{attribute 'GeneratedUsingTerminal: EK1122-0000-0018'}
{attribute addProperty BoxType "EK1122-0000-0018"}
{attribute addProperty Id "A_0060_AT2020_0250_0019_AT2020_0250A_0060_AT2020_0250_0019_AT2020_0250_BB71669A80Beckhoff_AT2xxxsub_EK1100EK1100_AB5A94672A_0001_AT2000_0233_0022AT2000_0D5D20CF80A_0002_AT2000_0233_0023AT2000_0D5D20CF80A_0003_AT2000_0233_0024AT2000_0D5D20CF80A_0004_AT2000_0250_0016AT2000_86175B4184A_0005_AT2000_0250_0017AT2000_86175B4184A_0006_AT2000_0250_0018AT2000_86175B4184A_0007_AT2000_0250_0019AT2000_86175B4184A_0008_AT2000_0250_0020AT2000_86175B4184A_0009_AT2000_0250_0021AT2000_86175B4184A_0010_AT2000_0250_0022AT2000_86175B4184A_0011_AT2000_0250_0023AT2000_86175B4184A_0012_AT2001_0250_0016AT2001_86175B4184A_0013_AT2001_0250_0017AT2001_86175B4184A_0014_AT2001_0250_0018AT2001_86175B4184A_0015_AT2001_0250_0019AT2001_86175B4184A_0016_AT2001_0250_0020AT2001_86175B4184A_0017_AT2001_0250_0022AT2001_86175B4184A_0018_AT2001_0250_0023AT2001_86175B4184A_0019_AT2001_0250_0024AT2001_86175B4184A_0020_AT2002_0249_0021AT2002_86175B4184A_0021_AT2002_0249_0022AT2002_86175B4184A_0022_AT2002_0249_0023AT2002_86175B4184A_0023_AT2002_0250_0022AT2002_86175B4184A_0024_AT2002_0250_0023AT2002_86175B4184A_0025_AT2002_0250_0024AT2002_86175B4184A_0026_AT2020_0250_0018AT2020_86175B4184A_0027_AT2020_0250_0021AT2020_86175B4184A_0028_AT2021_0250_0018AT2021_86175B4184A_0029_AT2021_0250_0020AT2021_86175B4184A_0030_AT2025_0250_0018AT2025_86175B4184A_0031_AT2026_0250_0021AT2026_86175B4184A_0032_AT2026_0250_0023AT2026_86175B4184A_0033_AT2040_0250_0018AT2040_86175B4184A_0034_AT2040_0250_0019AT2040_86175B4184A_0035_AT2040_0250_0020AT2040_86175B4184A_0036_AT2040_0250_0021A_0036_AT2040_0250_0021_991DCE0880A_0037_AT2040_0250_0022A_0037_AT2040_0250_0022_91A22A2880A_0038_AT2040_0250_0023A_0038_AT2040_0250_0023_51A62EE080A_0039_AT2040_0250_0024A_0039_AT2040_0250_0024_A5C6BC0680A_0040_AT2041_0250_0018A_0040_AT2041_0250_0018_C1FAE41E80A_0041_AT2041_0250_0019A_0041_AT2041_0250_0019_61D0A4BA80A_0042_AT2041_0250_0020A_0042_AT2041_0250_0020_CCFA41F280A_0043_AT2041_0250_0021A_0043_AT2041_0250_0021_389AD31480A_0044_AT2041_0250_0022A_0044_AT2041_0250_0022_C805DD5680A_0045_AT2041_0250_0023A_0045_AT2041_0250_0023_C359864080A_0046_AT2042_0250_0024A_0046_AT2042_0250_0024_89BF2BDD80A_0047_AT2050_0500_0016A_0047_AT2050_0500_0016_8100CFFD80A_0048_AT2050_0500_0017A_0048_AT2050_0500_0017_AD089BAB80A_0049_AT2050_0500_0018A_0049_AT2050_0500_0018_5979B14480A_0050_AT2050_0500_0019A_0050_AT2050_0500_0019_873C4A8380A_0051_AT2050_0500_0020A_0051_AT2050_0500_0020_09CCFFA280A_0052_AT2050_0500_0021A_0052_AT2050_0500_0021_D789046580A_0053_AT2050_0500_0022A_0053_AT2050_0500_0022_D1A4391280A_0054_AT2050_0500_0023A_0054_AT2050_0500_0023_206D3BB980A_0055_AT2050_0500_0024A_0055_AT2050_0500_0024_1FDD446180A_0056_AT2050_0501_0017A_0056_AT2050_0501_0017_33D5103780A_0057_AT2050_0501_0020A_0057_AT2050_0501_0020_3B6AF41780A_0058_AT2050_0501_0021A_0058_AT2050_0501_0021_4F11F47C80A_0061_AT2020_0250_0023_AT2020_0250A_0061_AT2020_0250_0023_AT2020_0250_BF05573080A_0062_AT2025_0250_0020_AT2025_0250A_0062_AT2025_0250_0020_AT2025_0250_1F2F179480A_0063_AT2025_0250_0022_AT2025_0250A_0063_AT2025_0250_0022_AT2025_0250_7A10824E80A_0064_AT2025_0250_0023_AT2025_0250A_0064_AT2025_0250_0023_AT2025_0250_1BD08B3080A_0065_AT2026_0250_0019_AT2026_0250A_0065_AT2026_0250_0019_AT2026_0250_37D8DF6680A_0066_AT2026_0250_0020_AT2026_0250A_0066_AT2026_0250_0020_AT2026_0250_3F673B4680A_0067_AT2026_0250_0022_AT2026_0250A_0067_AT2026_0250_0022_AT2026_0250_2DED6B0A80A_0068_AT2026_0250_0024_AT2026_0250A_0068_AT2026_0250_0024_AT2026_0250_E35FF58980A_0069_AT2050_0501_0019_AT2050_0501A_0069_AT2050_0501_0019_AT2050_0501_82BABB4A80A_0070_AT2050_0501_0022_AT2050_0501A_0070_AT2050_0501_0022_AT2050_0501_76DA29AC80A_0071_AT2050_0501_0023_AT2050_0501A_0071_AT2050_0501_0023_AT2050_0501_3753726880A_0072_AT2050_0501_0024_AT2050_0501A_0072_AT2050_0501_0024_AT2050_0501_977932CC80"}
{attribute addProperty CRC "2549082078"}
{attribute addProperty Size "5810"}
TYPE Beckhoff_AT2xxxEK1122_97EFE7DE EXTENDS EK1122_AB5A9467 :
STRUCT
	{attribute addProperty Name "A_0060_AT2020_0250_0019_AT2020_0250"}
	A_0060_AT2020_0250_0019_AT2020_0250 : A_0060_AT2020_0250_0019_AT2020_0250_BB71669A;
	{attribute addProperty Name "Beckhoff_AT2xxxsub_EK1100"}
	Beckhoff_AT2xxxsub_EK1100 : EK1100_AB5A9467;
	{attribute addProperty Name "A_0001_AT2000_0233_0022"}
	A_0001_AT2000_0233_0022 : AT2000_0D5D20CF;
	{attribute addProperty Name "A_0002_AT2000_0233_0023"}
	A_0002_AT2000_0233_0023 : AT2000_0D5D20CF;
	{attribute addProperty Name "A_0003_AT2000_0233_0024"}
	A_0003_AT2000_0233_0024 : AT2000_0D5D20CF;
	{attribute addProperty Name "A_0004_AT2000_0250_0016"}
	A_0004_AT2000_0250_0016 : AT2000_86175B41;
	{attribute addProperty Name "A_0005_AT2000_0250_0017"}
	A_0005_AT2000_0250_0017 : AT2000_86175B41;
	{attribute addProperty Name "A_0006_AT2000_0250_0018"}
	A_0006_AT2000_0250_0018 : AT2000_86175B41;
	{attribute addProperty Name "A_0007_AT2000_0250_0019"}
	A_0007_AT2000_0250_0019 : AT2000_86175B41;
	{attribute addProperty Name "A_0008_AT2000_0250_0020"}
	A_0008_AT2000_0250_0020 : AT2000_86175B41;
	{attribute addProperty Name "A_0009_AT2000_0250_0021"}
	A_0009_AT2000_0250_0021 : AT2000_86175B41;
	{attribute addProperty Name "A_0010_AT2000_0250_0022"}
	A_0010_AT2000_0250_0022 : AT2000_86175B41;
	{attribute addProperty Name "A_0011_AT2000_0250_0023"}
	A_0011_AT2000_0250_0023 : AT2000_86175B41;
	{attribute addProperty Name "A_0012_AT2001_0250_0016"}
	A_0012_AT2001_0250_0016 : AT2001_86175B41;
	{attribute addProperty Name "A_0013_AT2001_0250_0017"}
	A_0013_AT2001_0250_0017 : AT2001_86175B41;
	{attribute addProperty Name "A_0014_AT2001_0250_0018"}
	A_0014_AT2001_0250_0018 : AT2001_86175B41;
	{attribute addProperty Name "A_0015_AT2001_0250_0019"}
	A_0015_AT2001_0250_0019 : AT2001_86175B41;
	{attribute addProperty Name "A_0016_AT2001_0250_0020"}
	A_0016_AT2001_0250_0020 : AT2001_86175B41;
	{attribute addProperty Name "A_0017_AT2001_0250_0022"}
	A_0017_AT2001_0250_0022 : AT2001_86175B41;
	{attribute addProperty Name "A_0018_AT2001_0250_0023"}
	A_0018_AT2001_0250_0023 : AT2001_86175B41;
	{attribute addProperty Name "A_0019_AT2001_0250_0024"}
	A_0019_AT2001_0250_0024 : AT2001_86175B41;
	{attribute addProperty Name "A_0020_AT2002_0249_0021"}
	A_0020_AT2002_0249_0021 : AT2002_86175B41;
	{attribute addProperty Name "A_0021_AT2002_0249_0022"}
	A_0021_AT2002_0249_0022 : AT2002_86175B41;
	{attribute addProperty Name "A_0022_AT2002_0249_0023"}
	A_0022_AT2002_0249_0023 : AT2002_86175B41;
	{attribute addProperty Name "A_0023_AT2002_0250_0022"}
	A_0023_AT2002_0250_0022 : AT2002_86175B41;
	{attribute addProperty Name "A_0024_AT2002_0250_0023"}
	A_0024_AT2002_0250_0023 : AT2002_86175B41;
	{attribute addProperty Name "A_0025_AT2002_0250_0024"}
	A_0025_AT2002_0250_0024 : AT2002_86175B41;
	{attribute addProperty Name "A_0026_AT2020_0250_0018"}
	A_0026_AT2020_0250_0018 : AT2020_86175B41;
	{attribute addProperty Name "A_0027_AT2020_0250_0021"}
	A_0027_AT2020_0250_0021 : AT2020_86175B41;
	{attribute addProperty Name "A_0028_AT2021_0250_0018"}
	A_0028_AT2021_0250_0018 : AT2021_86175B41;
	{attribute addProperty Name "A_0029_AT2021_0250_0020"}
	A_0029_AT2021_0250_0020 : AT2021_86175B41;
	{attribute addProperty Name "A_0030_AT2025_0250_0018"}
	A_0030_AT2025_0250_0018 : AT2025_86175B41;
	{attribute addProperty Name "A_0031_AT2026_0250_0021"}
	A_0031_AT2026_0250_0021 : AT2026_86175B41;
	{attribute addProperty Name "A_0032_AT2026_0250_0023"}
	A_0032_AT2026_0250_0023 : AT2026_86175B41;
	{attribute addProperty Name "A_0033_AT2040_0250_0018"}
	A_0033_AT2040_0250_0018 : AT2040_86175B41;
	{attribute addProperty Name "A_0034_AT2040_0250_0019"}
	A_0034_AT2040_0250_0019 : AT2040_86175B41;
	{attribute addProperty Name "A_0035_AT2040_0250_0020"}
	A_0035_AT2040_0250_0020 : AT2040_86175B41;
	{attribute addProperty Name "A_0036_AT2040_0250_0021"}
	A_0036_AT2040_0250_0021 : A_0036_AT2040_0250_0021_991DCE08;
	{attribute addProperty Name "A_0037_AT2040_0250_0022"}
	A_0037_AT2040_0250_0022 : A_0037_AT2040_0250_0022_91A22A28;
	{attribute addProperty Name "A_0038_AT2040_0250_0023"}
	A_0038_AT2040_0250_0023 : A_0038_AT2040_0250_0023_51A62EE0;
	{attribute addProperty Name "A_0039_AT2040_0250_0024"}
	A_0039_AT2040_0250_0024 : A_0039_AT2040_0250_0024_A5C6BC06;
	{attribute addProperty Name "A_0040_AT2041_0250_0018"}
	A_0040_AT2041_0250_0018 : A_0040_AT2041_0250_0018_C1FAE41E;
	{attribute addProperty Name "A_0041_AT2041_0250_0019"}
	A_0041_AT2041_0250_0019 : A_0041_AT2041_0250_0019_61D0A4BA;
	{attribute addProperty Name "A_0042_AT2041_0250_0020"}
	A_0042_AT2041_0250_0020 : A_0042_AT2041_0250_0020_CCFA41F2;
	{attribute addProperty Name "A_0043_AT2041_0250_0021"}
	A_0043_AT2041_0250_0021 : A_0043_AT2041_0250_0021_389AD314;
	{attribute addProperty Name "A_0044_AT2041_0250_0022"}
	A_0044_AT2041_0250_0022 : A_0044_AT2041_0250_0022_C805DD56;
	{attribute addProperty Name "A_0045_AT2041_0250_0023"}
	A_0045_AT2041_0250_0023 : A_0045_AT2041_0250_0023_C3598640;
	{attribute addProperty Name "A_0046_AT2042_0250_0024"}
	A_0046_AT2042_0250_0024 : A_0046_AT2042_0250_0024_89BF2BDD;
	{attribute addProperty Name "A_0047_AT2050_0500_0016"}
	A_0047_AT2050_0500_0016 : A_0047_AT2050_0500_0016_8100CFFD;
	{attribute addProperty Name "A_0048_AT2050_0500_0017"}
	A_0048_AT2050_0500_0017 : A_0048_AT2050_0500_0017_AD089BAB;
	{attribute addProperty Name "A_0049_AT2050_0500_0018"}
	A_0049_AT2050_0500_0018 : A_0049_AT2050_0500_0018_5979B144;
	{attribute addProperty Name "A_0050_AT2050_0500_0019"}
	A_0050_AT2050_0500_0019 : A_0050_AT2050_0500_0019_873C4A83;
	{attribute addProperty Name "A_0051_AT2050_0500_0020"}
	A_0051_AT2050_0500_0020 : A_0051_AT2050_0500_0020_09CCFFA2;
	{attribute addProperty Name "A_0052_AT2050_0500_0021"}
	A_0052_AT2050_0500_0021 : A_0052_AT2050_0500_0021_D7890465;
	{attribute addProperty Name "A_0053_AT2050_0500_0022"}
	A_0053_AT2050_0500_0022 : A_0053_AT2050_0500_0022_D1A43912;
	{attribute addProperty Name "A_0054_AT2050_0500_0023"}
	A_0054_AT2050_0500_0023 : A_0054_AT2050_0500_0023_206D3BB9;
	{attribute addProperty Name "A_0055_AT2050_0500_0024"}
	A_0055_AT2050_0500_0024 : A_0055_AT2050_0500_0024_1FDD4461;
	{attribute addProperty Name "A_0056_AT2050_0501_0017"}
	A_0056_AT2050_0501_0017 : A_0056_AT2050_0501_0017_33D51037;
	{attribute addProperty Name "A_0057_AT2050_0501_0020"}
	A_0057_AT2050_0501_0020 : A_0057_AT2050_0501_0020_3B6AF417;
	{attribute addProperty Name "A_0058_AT2050_0501_0021"}
	A_0058_AT2050_0501_0021 : A_0058_AT2050_0501_0021_4F11F47C;
	{attribute addProperty Name "A_0061_AT2020_0250_0023_AT2020_0250"}
	A_0061_AT2020_0250_0023_AT2020_0250 : A_0061_AT2020_0250_0023_AT2020_0250_BF055730;
	{attribute addProperty Name "A_0062_AT2025_0250_0020_AT2025_0250"}
	A_0062_AT2025_0250_0020_AT2025_0250 : A_0062_AT2025_0250_0020_AT2025_0250_1F2F1794;
	{attribute addProperty Name "A_0063_AT2025_0250_0022_AT2025_0250"}
	A_0063_AT2025_0250_0022_AT2025_0250 : A_0063_AT2025_0250_0022_AT2025_0250_7A10824E;
	{attribute addProperty Name "A_0064_AT2025_0250_0023_AT2025_0250"}
	A_0064_AT2025_0250_0023_AT2025_0250 : A_0064_AT2025_0250_0023_AT2025_0250_1BD08B30;
	{attribute addProperty Name "A_0065_AT2026_0250_0019_AT2026_0250"}
	A_0065_AT2026_0250_0019_AT2026_0250 : A_0065_AT2026_0250_0019_AT2026_0250_37D8DF66;
	{attribute addProperty Name "A_0066_AT2026_0250_0020_AT2026_0250"}
	A_0066_AT2026_0250_0020_AT2026_0250 : A_0066_AT2026_0250_0020_AT2026_0250_3F673B46;
	{attribute addProperty Name "A_0067_AT2026_0250_0022_AT2026_0250"}
	A_0067_AT2026_0250_0022_AT2026_0250 : A_0067_AT2026_0250_0022_AT2026_0250_2DED6B0A;
	{attribute addProperty Name "A_0068_AT2026_0250_0024_AT2026_0250"}
	A_0068_AT2026_0250_0024_AT2026_0250 : A_0068_AT2026_0250_0024_AT2026_0250_E35FF589;
	{attribute addProperty Name "A_0069_AT2050_0501_0019_AT2050_0501"}
	A_0069_AT2050_0501_0019_AT2050_0501 : A_0069_AT2050_0501_0019_AT2050_0501_82BABB4A;
	{attribute addProperty Name "A_0070_AT2050_0501_0022_AT2050_0501"}
	A_0070_AT2050_0501_0022_AT2050_0501 : A_0070_AT2050_0501_0022_AT2050_0501_76DA29AC;
	{attribute addProperty Name "A_0071_AT2050_0501_0023_AT2050_0501"}
	A_0071_AT2050_0501_0023_AT2050_0501 : A_0071_AT2050_0501_0023_AT2050_0501_37537268;
	{attribute addProperty Name "A_0072_AT2050_0501_0024_AT2050_0501"}
	A_0072_AT2050_0501_0024_AT2050_0501 : A_0072_AT2050_0501_0024_AT2050_0501_977932CC;
END_STRUCT
END_TYPE

(* stored: Version 1.2.0.0, ProductVersion 3.1.4024.9
   DUT Beckhoff_AT2xxxEK1122_97EFE7DE: Id {6094b803-3a6b-4a6f-9303-7d98b0f11876} *)
